# EPICS substitutions: iocBoot/ioc13bmd/Pelco_CM6700.substitutions
file "$(IP)/ipApp/Db/Pelco_CM6700.db"
{
pattern
{P,       R,       PORT}
{13BMD:,  Pelco1,  serial12}
}

file "$(IP)/ipApp/Db/Pelco_CM6700_names.db"
{
pattern
{P,       R,       STR}
{13BMD:,  Pelco1,  ZRST}
{13BMD:,  Pelco1,  ONST}
{13BMD:,  Pelco1,  TWST}
{13BMD:,  Pelco1,  THST}
{13BMD:,  Pelco1,  FRST}
{13BMD:,  Pelco1,  FVST}
{13BMD:,  Pelco1,  SXST}
{13BMD:,  Pelco1,  SVST}
{13BMD:,  Pelco1,  EIST}
{13BMD:,  Pelco1,  NIST}
{13BMD:,  Pelco1,  TEST}
{13BMD:,  Pelco1,  ELST}
{13BMD:,  Pelco1,  TVST}
{13BMD:,  Pelco1,  TTST}
{13BMD:,  Pelco1,  FTST}
{13BMD:,  Pelco1,  FFST}
}
